{attribute 'linkalways'} 
{attribute 'no_explicit_call' := 'This FB is a CLASS and must be accessed using methods or properties'}
{attribute 'enable_dynamic_creation'}
FUNCTION_BLOCK _UINT EXTENDS DatatypeBase
VAR
	localData : UINT;
	activeData : REFERENCE TO UINT REF= localData;
END_VAR

PROPERTY PUBLIC Address : PVOID
GET
Address := ADR(activeData);
END_GET
END_PROPERTY

METHOD PUBLIC ClearReference
VAR_INPUT
END_VAR
activeData REF= localData;
END_METHOD

METHOD PUBLIC Clone : I_Datatype
VAR
    pClone : POINTER TO _UINT;
END_VAR
pClone := __NEW(_UINT(InitialValue := Value));
Clone := pClone^;
END_METHOD

METHOD FB_init : BOOL
VAR_INPUT
	bInitRetains : BOOL; // if TRUE, the retain variables are initialized (warm start / cold start)
	bInCopyCode : BOOL;  // if TRUE, the instance afterwards gets moved into the copy code (online change)
	InitialValue : UINT;
END_VAR
localData := InitialValue;
END_METHOD

PROPERTY PUBLIC IecType : T_MAXSTRING
GET
IecType := 'UINT';
END_GET
END_PROPERTY

METHOD PUBLIC MakeReferenceTo
VAR_INPUT
	ReferenceTarget : REFERENCE TO UINT;
END_VAR
activeData REF= ReferenceTarget;
END_METHOD

METHOD PUBLIC SerializeWith
VAR_INPUT
	Serializer : I_Serializer;
END_VAR
Serializer.AddUdint(activeData);
END_METHOD

PROPERTY PUBLIC Size : UDINT
GET
Size := SIZEOF(activeData);
END_GET
END_PROPERTY

METHOD TryDeserializeFrom : BOOL
VAR_INPUT
	Deserializer : I_Deserializer;
END_VAR
TryDeserializeFrom := Deserializer.TryGetUint(activeData);
END_METHOD

METHOD TryMakeReferenceTo : BOOL
VAR_INPUT
	Target : I_Datatype;
END_VAR
VAR
	pTargetData : POINTER TO UINT;
END_VAR
IF NOT (Target.IecType = IecType) THEN
	RETURN;
END_IF

pTargetData := Target.Address;
activeData REF= pTargetData^;
TryMakeReferenceTo := TRUE;
END_METHOD

PROPERTY PUBLIC Value : UINT
GET
Value := activeData;
END_GET
SET
activeData := Value;
END_SET
END_PROPERTY

END_FUNCTION_BLOCK

(* stored: Version 1.1.0.1, ProductVersion 3.1.4024.12
   POU _UINT: Id {cbed6cf7-fbf8-097c-0293-0e7f1c3f5467}, SpecialFunc None
   Folder Constructor: Id {b7e865a1-de9f-0ea8-18fd-e29ef0580957}
   Property Address: Id {22c7e2a6-d61f-0110-0341-9057da1fd006}
   Get Get: Id {7898a754-28c6-0cd8-1f19-a87a05a0cb89}
   Method ClearReference: Id {baf875f5-1f23-045a-3d3a-d0a7a2635b26}
   Method Clone: Id {2d944782-2ce6-050d-19bd-069bc8760853}
   Method FB_init: Id {d1ec7ebf-bb74-0a8f-11a3-1e265fb5d1fa}
   Property IecType: Id {c80358ad-9725-00b1-21f9-51d714de8890}
   Get Get: Id {2aeddd07-38df-08d7-2365-4a94eb18b542}
   Method MakeReferenceTo: Id {2af064f3-480e-0bca-2a47-db6bdc774210}
   Method SerializeWith: Id {5f5154f1-dfb8-0779-035e-90f3ccd5434b}
   Property Size: Id {818d689a-c1e5-0e2e-00c7-72cee1d29c58}
   Get Get: Id {f74b3f26-9c14-08a6-1d9e-5e5266d43f5f}
   Method TryDeserializeFrom: Id {964046c2-bce0-0078-0712-c6b8f5581b56}
   Method TryMakeReferenceTo: Id {052e8ae9-d393-02c4-0feb-8bd1204f1259}
   Property Value: Id {de8c7a46-b714-0d21-2f16-eba009ade7c8}
   Get Get: Id {ba0296e2-b2da-0c10-39df-84db5623f947}
   Set Set: Id {d73e9a79-7509-0f01-11c7-35ddcd43c48b} *)
